{attribute 'qualified_only'}
{attribute 'strict'}
TYPE test_state :
(
	IDLE,
	DATETIME2JD,
	EQ2HOR,
	DEG2RAD,
	RAD2DEG,
	JD2LST,
	ERROR
);
END_TYPE

(* stored: Version 1.1.0.1, ProductVersion 3.1.4024.12
   DUT test_state: Id {7e890740-17ec-420f-b803-923d73845ddd} *)
